KUKA KRL data list: A22_fls_global.dat

&ACCESS RV
&REL 1
&COMMENT V_1_4_1
DEFDAT A22_fls_global PUBLIC
;********************************
;Date: 07.11.2018
;Programmer: AIUT
;Description: Global positions
;********************************


ENDDAT
